(* Logix 5000 project; controller EuniceF_ICA9 vendor 1 type 14 code 150 rev 37.11; software revision 37.00 *)

TASK MainTask (continuous, watchdog 500 ms) : MainProgram

MODULES
   Local : vendor 1 type 14 code 150 (Compact 0, rev 37.11)
      Discrete_IO : Embedded (Compact 1, rev 3.1, Output RPI 20 ms)
      Analog_IO : Embedded (Compact 2, rev 1.1, Output RPI 80 ms)
      Counters : Embedded (Compact 3, rev 1.1, Output RPI 20 ms)
END_MODULES

VAR_GLOBAL   (* controller tags *)
   RUNNING : ALIAS FOR Local:1:O.Data.0;
   START : ALIAS FOR Local:1:I.Data.11;
   STOP : ALIAS FOR Local:1:I.Data.8;
   Timer1 : TIMER := (PRE := 10000);
END_VAR

PROGRAM MainProgram   (* main routine MainRoutine *)

ROUTINE MainRoutine   (* ladder *)
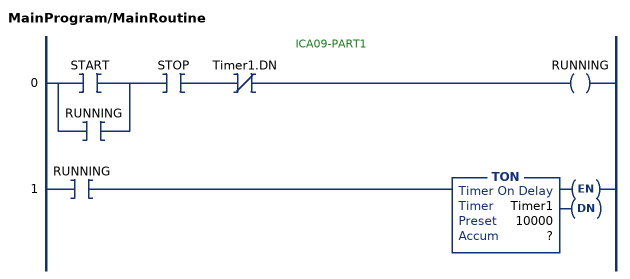
   // ICA09-PART1
   0: [XIC(START) ,XIC(RUNNING) ]XIC(STOP)XIO(Timer1.DN)OTE(RUNNING);
   1: XIC(RUNNING)TON(Timer1,?,?);
END_ROUTINE
END_PROGRAM
